(* CODESYS project visu_main_native.xml

Project tree, tasks and I/O mapping:
  visualisation VisuMain
*)

// /VisuMain
VISUALIZATION VisuMain  // 1024x768
END_VISUALIZATION
